# B&R Automation Studio project Stojan1
Automation Studio 4.2.9.65 SP

## Configuration Config1

CPU 5PPC2100.BY22-000, AutomationRuntime D4.26, Build 4.1.2, Vc V4.26.1

### Task classes (Cpu.sw)
```
Cyclic#1:
  ncsdcctrl <- ncsdcctrl.prg
  RdBlock_0 <- RdBlock_0.prg
Binaries: TCData, arconfig, asfw, ashwd, iomap, User, Role, sysconf
```

### IoMap.iom - 5PPC2100_BY22_000/IoMap.iom
```iecst
VAR_CONFIG
	::RdBlock_0:FltMtuRd[1] AT %IB."X20AP3131".RxByte1;
	::RdBlock_0:FltMtuRd[2] AT %IB."X20AP3131".RxByte2;
	::RdBlock_0:FltMtuRd[3] AT %IB."X20AP3131".RxByte3;
	::RdBlock_0:FltMtuRd[4] AT %IB."X20AP3131".RxByte4;
	::RdBlock_0:FltMtuRd[5] AT %IB."X20AP3131".RxByte5;
	::RdBlock_0:FltMtuRd[6] AT %IB."X20AP3131".RxByte6;
	::RdBlock_0:FltMtuRd[7] AT %IB."X20AP3131".RxByte7;
	::RdBlock_0:RBTrigDFT AT %IX."X20AP3131".RBTrigDFT;
	::RdBlock_0:TrigDFT AT %QX."X20AP3131".TrigDFT;
	::RdBlock_0:EnabEnergy AT %QX."X20AP3131".EnabEnergy;
	::RdBlock_0:FltMtuWr[0] AT %QB."X20AP3131".OutputSequence;
	RdBlock_0:FltMtuRd[0] AT %IB."X20AP3131".InputSequence;
END_VAR
```

## Configuration TestStand1

CPU , AutomationRuntime D3.10, Build 4.1.2

### Task classes (Cpu.sw)
```
Cyclic#1 (cycle 2000 us, tolerance 0 us):
  ncsdcctrl <- ncsdcctrl.prg
  RdBlock_0 <- RdBlock_0.prg
Cyclic#2 (cycle 20000 us, tolerance 20000 us):
  GearAxis01 <- Samples.GearAxis01.prg
  GearAxis02 <- Samples.GearAxis02.prg
DataObjects: Acp10sys
NcDataObjects: gAxis01a <- gAxis01obj.gAxis01a.dob, gAxis01i <- gAxis01obj.gAxis01i.dob, gAxis02a <- gAxis02obj.gAxis02a.dob, gAxis02i <- gAxis02obj.gAxis02i.dob, gAxis03a <- gAxis03obj.gAxis03a.dob, gAxis03i <- gAxis03obj.gAxis03i.dob, gAxis04a <- gAxis04obj.gAxis04a.dob, gAxis04i <- gAxis04obj.gAxis04i.dob
Binaries: ashwd, sysconf, asfw, arconfig, iomap, acp10map, acp10cfg
Libraries: Acp10_MC, brsystem, Acp10man, sys_lib, NcGlobal, Acp10par, Runtime, Acp10sdc, asstring, Acp10sim, astime, fileio, powerlnk, asieccon, asfltgen
```

### Hardware
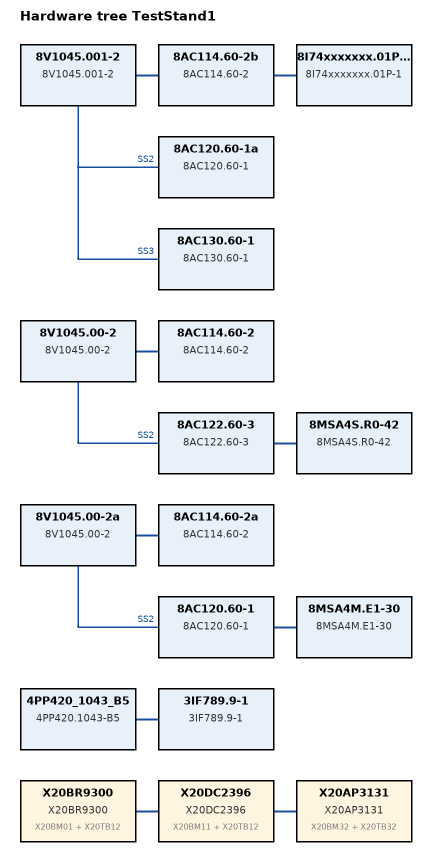
```
3IF789.9-1 : 3IF789.9-1 v1.1.3.1  [SS -> 4PP420_1043_B5.SS1]
  Connector IF2:
    EplEthInterfaceRedundant = 0
4PP420_1043_B5 : 4PP420.1043-B5 v1.0.0.0
  Connector IF5:
    ActivateDevice = 1
  TimerDeviceType = EPLX2X
  TimerDevice = 3IF789.9-1.IF2
  TaskClassIdleTime = 2000
  Cyclic1Duration = 2000
  Cyclic1Tolerance = 0
  Cyclic1Output = 1
  Cyclic2Duration = 20000
  Cyclic2Tolerance = 20000
  Cyclic3Duration = 50000
  Cyclic3Tolerance = 50000
  Cyclic4Duration = 100000
  Cyclic4Tolerance = 100000
  Cyclic5Duration = 200000
  Cyclic5Tolerance = 200000
  Cyclic6Duration = 500000
  Cyclic6Tolerance = 500000
  Cyclic7Duration = 1000000
  Cyclic7Tolerance = 1000000
  Cyclic8Duration = 10000
  Cyclic8Tolerance = 30000000
  EthernetHostName = stojan1
8AC114.60-2 : 8AC114.60-2 v1.0.0.8  [SS -> 8V1045.00-2.SS1; PLK1 -> 3IF789.9-1.IF2 (NodeNumber=1); PLK2 -> 8AC114.60-2a.PLK1 (NodeNumber=1)]
8AC114.60-2a : 8AC114.60-2 v1.0.0.8  [SS -> 8V1045.00-2a.SS1; PLK1 -> 8AC114.60-2.PLK2 (NodeNumber=2); PLK2 -> 8AC114.60-2b.PLK1 (NodeNumber=2)]
8AC114.60-2b : 8AC114.60-2 v1.0.0.8  [SS -> 8V1045.001-2.SS1; PLK1 -> 8AC114.60-2a.PLK2 (NodeNumber=3); PLK2 -> 8I74xxxxxxx.01P-1.PLK1 (NodeNumber=3)]
8AC120.60-1 : 8AC120.60-1 v1.0.0.2  [SS -> 8V1045.00-2a.SS2]
8AC120.60-1a : 8AC120.60-1 v1.0.0.2  [SS -> 8V1045.001-2.SS2]
8AC122.60-3 : 8AC122.60-3 v1.0.0.2  [SS -> 8V1045.00-2.SS2]
8AC130.60-1 : 8AC130.60-1 v1.0.0.3  [SS -> 8V1045.001-2.SS3]
8I74xxxxxxx.01P-1 : 8I74xxxxxxx.01P-1 v1.2.0.1  [PLK1 -> 8AC114.60-2b.PLK2 (NodeNumber=4)]
  Supervision = off
  CTT = 3
  AUT = 1
  NPR = 75
  COS = 80
  UNS = 400
  NCR = 19
  NSP = 1395
  RSA = 11302
  LFA = 4842
8MSA4M.E1-30 : 8MSA4M.E1-30 v1.0.0.0  [EC -> 8AC120.60-1.EC; MT -> 8V1045.00-2a.MT1]
8MSA4S.R0-42 : 8MSA4S.R0-42 v1.0.0.0  [EC -> 8AC122.60-3.EC; MT -> 8V1045.00-2.MT1]
8V1045.00-2 : 8V1045.00-2 v1.0.0.2
  BothEndSwitchesAreNormallyOpen_r1 = on
  QuickStopIsNormallyOpen_r1 = on
8V1045.00-2a : 8V1045.00-2 v1.0.0.2
  BothEndSwitchesAreNormallyOpen_r1 = on
  QuickStopIsNormallyOpen_r1 = on
8V1045.001-2 : 8V1045.001-2 v1.0.0.0
  BothEndSwitchesAreNormallyOpen_r1 = on
  QuickStopIsNormallyOpen_r1 = on
X20AP3131 : X20AP3131 v1.0.1.0  [SS1 -> X20TB32.SS; SL -> X20BM32.SL1]
  Supervision = off
  EnergyUnit = 1Ws
  VoltageLimit = off
  DisPFmeanT = off
  DisPmeanT = off
  DisQmeanT = off
  DisSmeanT = off
  DisAcEnT = off
  DisReacEnT = off
  DisAppEnT = off
  FlatStreamActivate = on
  InputMTU = 23byte
X20BM01 : X20BM01 v1.0.1.1
X20BM11 : X20BM11 v1.0.0.1  [X2X1 -> X20BM01.X2X2]
X20BM32 : X20BM32 v1.0.0.1  [X2X1 -> X20BM11.X2X2]
X20BR9300 : X20BR9300 v1.0.3.0  [SS1 -> X20TB12.SS; SL -> X20BM01.SL1; X2X1 -> 3IF789.9-1.IF1]
  Supervision = off
X20DC2396 : X20DC2396 v1.0.2.1  [SS1 -> X20TB12a.SS; SL -> X20BM11.SL1]
  Supervision = off
X20TB12 : X20TB12 v1.0.0.0
X20TB12a : X20TB12 v1.0.0.0
X20TB32 : X20TB32 v1.0.0.1
```

### IoMap.iom - 4PP420_1043_B5/IoMap.iom
```iecst
(********************************************************************
 * COPYRIGHT -- Bernecker + Rainer
 ********************************************************************
 * File: IoMap.iom
 * Author: necidj
 * Created: March 11, 2014
 ********************************************************************
 * IO mapping file
 ********************************************************************)
VAR_CONFIG
	Cyclic#1.gAxis04_DrvIf.iLifeCnt AT %IB."8I74xxxxxxx.01P-1".SDC_LifeCnt;
	Cyclic#1.gAxis04_DrvIf.iDrvOK AT %IX."8I74xxxxxxx.01P-1".ETAD_Input_Bool_02;
	Cyclic#1.gAxis04_DrvIf.oSetTime AT %QW."8I74xxxxxxx.01P-1".SDC_SetTime;
	Cyclic#1.gAxis04_DrvIf.oSetPos AT %QW."8I74xxxxxxx.01P-1".LFRD_Output;
	Cyclic#1.gAxis04_DiDoIf.iLifeCntDriveReady AT %IB."8I74xxxxxxx.01P-1".SDC_LifeCnt;
	Cyclic#1.gAxis04_DiDoIf.iLifeCntDriveEnable AT %IB."8I74xxxxxxx.01P-1".SDC_LifeCnt;
	Cyclic#1.gAxis04_DiDoIf.oDriveEnable AT %QX."8I74xxxxxxx.01P-1".CMDD_Output_Bool_00;
	Cyclic#1.gAxis04_ModuleOk AT %QX."8I74xxxxxxx.01P-1".CMDD_Output_Bool_01;
	Cyclic#1.gAxis04_ModuleOk AT %QX."8I74xxxxxxx.01P-1".CMDD_Output_Bool_02;
	Cyclic#1.gAxis04_ModuleOk AT %IX."8I74xxxxxxx.01P-1".ModuleOk;
	Cyclic#1.gAxis04_DiDoIf.oDriveEnable AT %QX."8I74xxxxxxx.01P-1".CMDD_Output_Bool_03;
	Cyclic#1.gAxis04_DiDoIf.iDriveReady AT %IX."8I74xxxxxxx.01P-1".ETAD_Input_Bool_02;
	gAxis04_DrvIf.oBrake AT %QX."8I74xxxxxxx.01P-1".OL1R_Output_Bool_02;
	gAxis04_EncIf.iActPos AT %IW."X20DC2396".Encoder01;
	gAxis04_EncIf.iEncOK AT %IX."X20DC2396".ModuleOk;
	::RdBlock_0:FltMtuRd[1] AT %IB."X20AP3131".RxByte1;
	::RdBlock_0:FltMtuRd[2] AT %IB."X20AP3131".RxByte2;
	::RdBlock_0:FltMtuRd[3] AT %IB."X20AP3131".RxByte3;
	::RdBlock_0:FltMtuRd[4] AT %IB."X20AP3131".RxByte4;
	::RdBlock_0:FltMtuRd[5] AT %IB."X20AP3131".RxByte5;
	::RdBlock_0:FltMtuRd[6] AT %IB."X20AP3131".RxByte6;
	::RdBlock_0:FltMtuRd[7] AT %IB."X20AP3131".RxByte7;
	::RdBlock_0:FltMtuRd[8] AT %IB."X20AP3131".RxByte8;
	::RdBlock_0:FltMtuRd[9] AT %IB."X20AP3131".RxByte9;
	::RdBlock_0:FltMtuRd[10] AT %IB."X20AP3131".RxByte10;
	::RdBlock_0:FltMtuRd[11] AT %IB."X20AP3131".RxByte11;
	::RdBlock_0:FltMtuRd[12] AT %IB."X20AP3131".RxByte12;
	::RdBlock_0:FltMtuRd[13] AT %IB."X20AP3131".RxByte13;
	::RdBlock_0:FltMtuRd[14] AT %IB."X20AP3131".RxByte14;
	::RdBlock_0:FltMtuRd[15] AT %IB."X20AP3131".RxByte15;
	::RdBlock_0:FltMtuRd[16] AT %IB."X20AP3131".RxByte16;
	::RdBlock_0:FltMtuRd[17] AT %IB."X20AP3131".RxByte17;
	::RdBlock_0:FltMtuRd[18] AT %IB."X20AP3131".RxByte18;
	::RdBlock_0:FltMtuRd[19] AT %IB."X20AP3131".RxByte19;
	::RdBlock_0:FltMtuRd[20] AT %IB."X20AP3131".RxByte20;
	::RdBlock_0:FltMtuRd[21] AT %IB."X20AP3131".RxByte21;
	::RdBlock_0:FltMtuRd[22] AT %IB."X20AP3131".RxByte22;
	::RdBlock_0:RBTrigDFT AT %IX."X20AP3131".RBTrigDFT;
	::RdBlock_0:TrigDFT AT %QX."X20AP3131".TrigDFT;
	::RdBlock_0:EnabEnergy AT %QX."X20AP3131".EnabEnergy;
	RdBlock_0:FltMtuRd[23]  AT %IB."X20AP3131".RxByte23;
	::RdBlock_0:FltMtuWr[0] AT %QB."X20AP3131".OutputSequence;
	RdBlock_0:FltMtuRd[0]  AT %IB."X20AP3131".InputSequence;
END_VAR
```

### Acp10cfg.ncc - 4PP420_1043_B5/Motion/Acp10cfg.ncc
```
NcConfiguration (Version=2.42.0, NcSwId=Acp10)
  ACP10CF1_typ:
    cnt_nettrc_rec_drive = 1500
    bufsize_trace_upload = 1200
    tc_nc_man_task = Cyclic #1
    glob_pv_as_ncobject = Yes
    ncsys_dl_broadcast = Yes
    ncsys_dl_acp_reset = Yes
    safemc_log_err_to_ax = Yes
    network_init:
      ncsw_init_execute = Yes
      automatic_execute = No
      node_nr_warning = Yes
      net_err_before_ncact = Yes
    nettrc:
      enter_parsecrec = Yes
      enter_ncaction = Yes
      save_ring_startidx = Yes
    cam_prof_download:
      cam_dat_dl_parallel = No
      tc_cam_dl_parallel = Task class for NC Manager task
    plk_if[0]:
      if_name = SL1.SS1.IF2
      tc_CycDat_PLCopen = Task class for NC Manager task
      mc_broadcast_extdat = No
    sdc_if[0]:
      if_name = SDC_IF1
      mc_broadcast_size = 800
      mc_broadcast_extdat = No
```

### Acp10map.ncm - 4PP420_1043_B5/Motion/Acp10map.ncm
```
NcMapping (NcSwId=Acp10)
  NcObject gAxis01 (ModuleId=8V1045.00-2, Type=ncAXIS, Channel=1, AcoposSimulation=Standard, InitParameter=gAxis01i, AcoposParameter=gAxis01a, Disabled=FALSE, ModuleDisabled=FALSE)
  NcObject 8V1045.00-2_ncV_AXIS1 (ModuleId=8V1045.00-2, Type=ncV_AXIS, Channel=1, Disabled=TRUE, ModuleDisabled=FALSE)
  NcObject gAxis02 (ModuleId=8V1045.00-2a, Type=ncAXIS, Channel=1, AcoposSimulation=Standard, InitParameter=gAxis02i, AcoposParameter=gAxis02a, Disabled=FALSE, ModuleDisabled=FALSE)
  NcObject 8V1045.00-2a_ncV_AXIS1 (ModuleId=8V1045.00-2a, Type=ncV_AXIS, Channel=1, Disabled=TRUE, ModuleDisabled=FALSE)
  NcObject gAxis03 (ModuleId=8V1045.001-2, Type=ncAXIS, Channel=1, AcoposSimulation=Off, InitParameter=gAxis03i, AcoposParameter=gAxis03a, Disabled=FALSE, ModuleDisabled=FALSE)
  NcObject 8V1045.001-2_ncV_AXIS1 (ModuleId=8V1045.001-2, Type=ncV_AXIS, Channel=1, Disabled=TRUE, ModuleDisabled=FALSE)
  NcObject gAxis04 (ModuleId=8I74xxxxxxx.01P-1, ModuleAddress=SDC_IF1.ST1, Type=ncAXIS, Channel=1, AcoposSimulation=Off, InitParameter=gAxis04i, AcoposParameter=gAxis04a, Disabled=FALSE, ModuleDisabled=FALSE)
```

## Logical view

Binary libraries used (declarations not repeated): operator, runtime, astime, AsIecCon, brsystem, sys_lib, asstring, Acp10man 2.43.1, Acp10par 2.43.1, NcGlobal 2.43.1, Acp10_MC 2.43.1, Acp10sdc 2.43.1, Acp10sim 2.43.1, AsFltGen

### Global.var - Global variables
```iecst
(********************************************************************
 * COPYRIGHT -- Bernecker + Rainer
 ********************************************************************
 * File: Global.var
 * Author: necidj
 * Created: March 11, 2014
 ********************************************************************
 * Global variables of project TestStandBasic
 ********************************************************************)
VAR
	gAxis01 : ACP10AXIS_typ;
	gAxis02 : ACP10AXIS_typ;
	gAxis03 : ACP10AXIS_typ;
	gAxis04 : ACP10AXIS_typ;
	gAxis04_HW : SdcHwCfg_typ := (0);
	gAxis04_EncIf : SdcEncIf16_typ := (0);
	gAxis04_DrvIf : SdcDrvIf16_typ := (0);
	gAxis04_DiDoIf : SdcDiDoIf_typ := (0);
	gAxis04_ModuleOk : BOOL := 0;
END_VAR
```


### Package Logical/gAxis01obj - gAxis01obj

- Data object Logical/gAxis01obj/gAxis01a (Apt) (no source held here)

### Data object Logical/gAxis01obj/gAxis01i (Ax)

#### gAxis01i.ax
```
InitParameter (Version=2.43.1, NcSwId=ACP10)
  ACP10AXIS_typ:
    dig_in:
      level:
        reference = ncACTIV_HI
        pos_hw_end = ncACTIV_HI
        neg_hw_end = ncACTIV_HI
        trigger1 = ncACTIV_HI
        trigger2 = ncACTIV_HI
    encoder_if:
      parameter:
        count_dir = ncSTANDARD
        scaling:
          load:
            units = 1000
            rev_motor = 1
    limit:
      parameter:
        v_pos = 10000.0
        v_neg = 10000.0
        a1_pos = 50000.0
        a2_pos = 50000.0
        a1_neg = 50000.0
        a2_neg = 50000.0
        t_jolt = 0.0
        t_in_pos = 0.0
        pos_sw_end = 8388607
        neg_sw_end = -8388608
        ds_warning = 500.0
        ds_stop = 1000.0
        a_stop = 1.0e+30
        dv_stop = 0.0
        dv_stop_mode = ncOFF
    controller:
      mode = ncPOSITION
      position:
        kv = 440.0
        tn = 0.0
        t_predict = 0.0004
        t_total = 0.0004
        p_max = 1.0e+30
        i_max = 0.0
      speed:
        kv = 3.5
        tn = 0.0
        t_filter = 0.0012
        isq_filter1:
          type = ncNOTCH
          a0 = 2485.32
          a1 = 400.0
          b0 = 0.0
          b1 = 0.0
          b2 = 0.0
          c0_par_id = 0
          c1_par_id = 0
        isq_filter2:
          type = ncOFF
          a0 = 0.0
          a1 = 0.0
          b0 = 0.0
          b1 = 0.0
          b2 = 0.0
          c0_par_id = 0
          c1_par_id = 0
        isq_filter3:
          type = ncOFF
          a0 = 0.0
          a1 = 0.0
          b0 = 0.0
          b1 = 0.0
          b2 = 0.0
          c0_par_id = 0
          c1_par_id = 0
      uf:
        type = ncLINEAR
        auto_config = ncMOTOR_PAR
        u0 = 0.0
        un = 0.0
        fn = 50.0
        k_f_slip = 0.0
      ff:
        torque_load = 0.0
        torque_pos = 0.0
        torque_neg = 0.0
        kv_torque = 0.0
        inertia = 0.0
        t_filter_a = 0.0
    move:
      stop:
        parameter[0]:
          decel_ramp = ncA_LIMIT
          controller = ncON
        parameter[1]:
          decel_ramp = ncA_LIMIT
          controller = ncON
        parameter[2]:
          decel_ramp = ncA_LIMIT
          controller = ncON
        parameter[3]:
          decel_ramp = ncA_LIMIT
          controller = ncON
        quickstop:
          decel_ramp = ncA_LIMIT
        drive_error:
          decel_ramp = ncA_LIMIT
      homing:
        parameter:
          s = 0
          v_switch = 5000.0
          v_trigger = 500.0
          a = 50000.0
          mode = ncDIRECT
          edge_sw = ncPOSITIVE
          start_dir = ncPOSITIVE
          trigg_dir = ncPOSITIVE
          ref_pulse = ncOFF
          fix_dir = ncOFF
          tr_s_block = 0.0
          torque_lim = 0.0
          ds_block = 0.0
          ds_stop = 0.0
      basis:
        parameter:
          v_pos = 5000.0
          v_neg = 5000.0
          a1_pos = 50000.0
          a2_pos = 50000.0
          a1_neg = 50000.0
          a2_neg = 50000.0
    message:
      text:
        parameter:
          format = ncBREAK
          columns = 80
          data_modul = acp10etxen
```

### Package Logical/gAxis02obj - gAxis02obj

### Data object Logical/gAxis02obj/gAxis02a (Apt)

#### gAxis02a.apt
```
AcoposParameterTable:
  Root Parameters
```

### Data object Logical/gAxis02obj/gAxis02i (Ax)

#### gAxis02i.ax
```
InitParameter (Version=2.43.1, NcSwId=ACP10)
  ACP10AXIS_typ:
    dig_in:
      level:
        reference = ncACTIV_HI
        pos_hw_end = ncACTIV_HI
        neg_hw_end = ncACTIV_HI
        trigger1 = ncACTIV_HI
        trigger2 = ncACTIV_HI
    encoder_if:
      parameter:
        count_dir = ncSTANDARD
        scaling:
          load:
            units = 1000
            rev_motor = 1
    limit:
      parameter:
        v_pos = 10000.0
        v_neg = 10000.0
        a1_pos = 50000.0
        a2_pos = 50000.0
        a1_neg = 50000.0
        a2_neg = 50000.0
        t_jolt = 0.0
        t_in_pos = 0.0
        pos_sw_end = 8388607
        neg_sw_end = -8388608
        ds_warning = 500.0
        ds_stop = 1000.0
        a_stop = 1.0e+30
        dv_stop = 0.0
        dv_stop_mode = ncOFF
    controller:
      mode = ncPOSITION
      position:
        kv = 40.0
        tn = 0.0
        t_predict = 0.0004
        t_total = 0.0004
        p_max = 1.0e+30
        i_max = 0.0
      speed:
        kv = 1.2
        tn = 0.0
        t_filter = 0.0004
        isq_filter1:
          type = ncNOTCH
          a0 = 1771.04
          a1 = 400.0
          b0 = 0.0
          b1 = 0.0
          b2 = 0.0
          c0_par_id = 0
          c1_par_id = 0
        isq_filter2:
          type = ncOFF
          a0 = 0.0
          a1 = 0.0
          b0 = 0.0
          b1 = 0.0
          b2 = 0.0
          c0_par_id = 0
          c1_par_id = 0
        isq_filter3:
          type = ncOFF
          a0 = 0.0
          a1 = 0.0
          b0 = 0.0
          b1 = 0.0
          b2 = 0.0
          c0_par_id = 0
          c1_par_id = 0
      uf:
        type = ncLINEAR
        auto_config = ncMOTOR_PAR
        u0 = 0.0
        un = 0.0
        fn = 50.0
        k_f_slip = 0.0
      ff:
        torque_load = 0.0
        torque_pos = 0.0
        torque_neg = 0.0
        kv_torque = 0.0
        inertia = 0.0
        t_filter_a = 0.0
    move:
      stop:
        parameter[0]:
          decel_ramp = ncA_LIMIT
          controller = ncON
        parameter[1]:
          decel_ramp = ncA_LIMIT
          controller = ncON
        parameter[2]:
          decel_ramp = ncA_LIMIT
          controller = ncON
        parameter[3]:
          decel_ramp = ncA_LIMIT
          controller = ncON
        quickstop:
          decel_ramp = ncA_LIMIT
        drive_error:
          decel_ramp = ncA_LIMIT
      homing:
        parameter:
          s = 0
          v_switch = 5000.0
          v_trigger = 500.0
          a = 50000.0
          mode = ncDIRECT
          edge_sw = ncPOSITIVE
          start_dir = ncPOSITIVE
          trigg_dir = ncPOSITIVE
          ref_pulse = ncOFF
          fix_dir = ncOFF
          tr_s_block = 0.0
          torque_lim = 0.0
          ds_block = 0.0
          ds_stop = 0.0
      basis:
        parameter:
          v_pos = 5000.0
          v_neg = 5000.0
          a1_pos = 50000.0
          a2_pos = 50000.0
          a1_neg = 50000.0
          a2_neg = 50000.0
    message:
      text:
        parameter:
          format = ncBREAK
          columns = 80
          data_modul = acp10etxen
```

### Package Logical/gAxis03obj - gAxis03obj

- Data object Logical/gAxis03obj/gAxis03a (Apt) (no source held here)

### Data object Logical/gAxis03obj/gAxis03i (Ax)

#### gAxis03i.ax
```
InitParameter (Version=2.42.1, NcSwId=ACP10)
  ACP10AXIS_typ:
    dig_in:
      level:
        reference = ncACTIV_HI
        pos_hw_end = ncACTIV_HI
        neg_hw_end = ncACTIV_HI
        trigger1 = ncACTIV_HI
        trigger2 = ncACTIV_HI
    encoder_if:
      parameter:
        count_dir = ncSTANDARD
        scaling:
          load:
            units = 1000
            rev_motor = 1
    limit:
      parameter:
        v_pos = 10000.0
        v_neg = 10000.0
        a1_pos = 50000.0
        a2_pos = 50000.0
        a1_neg = 50000.0
        a2_neg = 50000.0
        t_jolt = 0.0
        t_in_pos = 0.0
        pos_sw_end = 8388607
        neg_sw_end = -8388608
        ds_warning = 500.0
        ds_stop = 1000.0
        a_stop = 1.0e+30
        dv_stop = 0.0
        dv_stop_mode = ncOFF
    controller:
      mode = ncPOSITION + ncFF
      position:
        kv = 520.0
        tn = 0.0
        t_predict = 0.0004
        t_total = 0.0004
        p_max = 1.0e+30
        i_max = 0.0
      speed:
        kv = 0.2
        tn = 0.0
        t_filter = 0.0
        isq_filter1:
          type = ncOFF
          a0 = 0.0
          a1 = 0.0
          b0 = 0.0
          b1 = 0.0
          b2 = 0.0
          c0_par_id = 0
          c1_par_id = 0
        isq_filter2:
          type = ncOFF
          a0 = 0.0
          a1 = 0.0
          b0 = 0.0
          b1 = 0.0
          b2 = 0.0
          c0_par_id = 0
          c1_par_id = 0
        isq_filter3:
          type = ncOFF
          a0 = 0.0
          a1 = 0.0
          b0 = 0.0
          b1 = 0.0
          b2 = 0.0
          c0_par_id = 0
          c1_par_id = 0
      uf:
        type = ncLINEAR
        auto_config = ncMOTOR_PAR
        u0 = 0.0
        un = 0.0
        fn = 50.0
        k_f_slip = 0.0
      ff:
        torque_load = 0.0
        torque_pos = 0.0287764
        torque_neg = 0.0287767
        kv_torque = 0.00626887
        inertia = 0.00413145
        t_filter_a = 0.0
    move:
      stop:
        parameter[0]:
          decel_ramp = ncA_LIMIT
          controller = ncON
        parameter[1]:
          decel_ramp = ncA_LIMIT
          controller = ncON
        parameter[2]:
          decel_ramp = ncA_LIMIT
          controller = ncON
        parameter[3]:
          decel_ramp = ncA_LIMIT
          controller = ncON
        quickstop:
          decel_ramp = ncA_LIMIT
        drive_error:
          decel_ramp = ncA_LIMIT
      homing:
        parameter:
          s = 0
          v_switch = 5000.0
          v_trigger = 500.0
          a = 50000.0
          mode = ncDIRECT
          edge_sw = ncPOSITIVE
          start_dir = ncPOSITIVE
          trigg_dir = ncPOSITIVE
          ref_pulse = ncOFF
          fix_dir = ncOFF
          tr_s_block = 0.0
          torque_lim = 0.0
          ds_block = 0.0
          ds_stop = 0.0
      basis:
        parameter:
          v_pos = 5000.0
          v_neg = 5000.0
          a1_pos = 50000.0
          a2_pos = 50000.0
          a1_neg = 50000.0
          a2_neg = 50000.0
    message:
      text:
        parameter:
          format = ncBREAK
          columns = 80
          data_modul = acp10etxen
```

### Package Logical/gAxis04obj - gAxis04obj

### Data object Logical/gAxis04obj/gAxis04a (Apt)

#### gAxis04a.apt
```
AcoposParameterTable:
  Root Parameters:
    230 = PCTRL_S_SET (Name=PCTRL_S_ACT_PARID)
    64201 = 546116,666666667 (Name=SERVO_V_MAX_OUTPUT)
    90 = 77 (Name=BRAKE_MODE)  // Motor holding brake: Mode
```

### Data object Logical/gAxis04obj/gAxis04i (Ax)

#### gAxis04i.ax
```
InitParameter (Version=2.42.1, NcSwId=ACP10)
  ACP10AXIS_typ:
    dig_in:
      level:
        reference = ncACTIV_HI
        pos_hw_end = ncACTIV_HI
        neg_hw_end = ncACTIV_HI
        trigger1 = ncACTIV_HI
        trigger2 = ncACTIV_HI
    encoder_if:
      parameter:
        count_dir = ncSTANDARD
        scaling:
          load:
            units = 1000
            rev_motor = 1
    limit:
      parameter:
        v_pos = 10000.0
        v_neg = 10000.0
        a1_pos = 50000.0
        a2_pos = 50000.0
        a1_neg = 50000.0
        a2_neg = 50000.0
        t_jolt = 0.0
        t_in_pos = 0.0
        pos_sw_end = 8388607
        neg_sw_end = -8388608
        ds_warning = 500.0
        ds_stop = 1000.0
        a_stop = 1.0e+30
        dv_stop = 0.0
        dv_stop_mode = ncOFF
    controller:
      mode = ncPOSITION
      position:
        kv = 50.0
        tn = 0.0
        t_predict = 0.01
        t_total = 0.01
        p_max = 10000.0
        i_max = 0.0
      speed:
        kv = 2.0
        tn = 0.0
        t_filter = 0.0
        isq_filter1:
          type = ncOFF
          a0 = 0.0
          a1 = 0.0
          b0 = 0.0
          b1 = 0.0
          b2 = 0.0
          c0_par_id = 0
          c1_par_id = 0
        isq_filter2:
          type = ncOFF
          a0 = 0.0
          a1 = 0.0
          b0 = 0.0
          b1 = 0.0
          b2 = 0.0
          c0_par_id = 0
          c1_par_id = 0
        isq_filter3:
          type = ncOFF
          a0 = 0.0
          a1 = 0.0
          b0 = 0.0
          b1 = 0.0
          b2 = 0.0
          c0_par_id = 0
          c1_par_id = 0
      uf:
        type = ncLINEAR
        auto_config = ncMOTOR_PAR
        u0 = 0.0
        un = 0.0
        fn = 50.0
        k_f_slip = 0.0
      ff:
        torque_load = 0.0
        torque_pos = 0.0
        torque_neg = 0.0
        kv_torque = 0.0
        inertia = 0.0
        t_filter_a = 0.0
    move:
      stop:
        parameter[0]:
          decel_ramp = ncA_LIMIT
          controller = ncON
        parameter[1]:
          decel_ramp = ncA_LIMIT
          controller = ncON
        parameter[2]:
          decel_ramp = ncA_LIMIT
          controller = ncON
        parameter[3]:
          decel_ramp = ncA_LIMIT
          controller = ncON
        quickstop:
          decel_ramp = ncA_LIMIT
        drive_error:
          decel_ramp = ncA_LIMIT
      homing:
        parameter:
          s = 0
          v_switch = 5000.0
          v_trigger = 500.0
          a = 50000.0
          mode = ncDIRECT
          edge_sw = ncPOSITIVE
          start_dir = ncPOSITIVE
          trigg_dir = ncPOSITIVE
          ref_pulse = ncOFF
          fix_dir = ncOFF
          tr_s_block = 0.0
          torque_lim = 0.0
          ds_block = 0.0
          ds_stop = 0.0
      basis:
        parameter:
          v_pos = 5000.0
          v_neg = 5000.0
          a1_pos = 50000.0
          a2_pos = 50000.0
          a1_neg = 50000.0
          a2_neg = 50000.0
    message:
      text:
        parameter:
          format = ncBREAK
          columns = 80
          data_modul = acp10etxen
```

### Program Logical/ncsdcctrl (IEC)

#### ncsdcctrlCyclic.st
```iecst
(********************************************************************
 * COPYRIGHT -- Bernecker + Rainer
 ********************************************************************
 * Program: ncsdcctrl
 * File: ncsdcctrlCyclic.st
 * Author: necidj
 * Created: March 11, 2014
 ********************************************************************
 * Implementation of program ncsdcctrl
 ********************************************************************)

PROGRAM _CYCLIC

(* ### BEGIN gAxis04 ### *)

(* life counter emulation of digital inputs *)
 gAxis04_DiDoIf.iLifeCntReference := gAxis04_DiDoIf.iLifeCntReference + 1;
 gAxis04_DiDoIf.iLifeCntNegHwEnd  := gAxis04_DiDoIf.iLifeCntNegHwEnd  + 1;
 gAxis04_DiDoIf.iLifeCntPosHwEnd  := gAxis04_DiDoIf.iLifeCntPosHwEnd  + 1;

(* ### END gAxis04 ### *)

END_PROGRAM
```

#### ncsdcctrlInit.st
```iecst
(********************************************************************
 * COPYRIGHT -- Bernecker + Rainer
 ********************************************************************
 * Program: ncsdcctrl
 * File: ncsdcctrlInit.st
 * Author: necidj
 * Created: March 11, 2014
 ********************************************************************
 * Implementation of program ncsdcctrl
 ********************************************************************)

PROGRAM _INIT

(* ### BEGIN gAxis04 ### *)

(* initialize variables *)
 gAxis04_HW.DrvIf_Typ := ncSDC_DRVSERVO16;
 strcpy( ADR(gAxis04_HW.DrvIf_Name[0]), ADR('gAxis04_DrvIf') );
 gAxis04_HW.DiDoIf_Typ := ncSDC_DIDO;
 strcpy( ADR(gAxis04_HW.DiDoIf_Name[0]), ADR('gAxis04_DiDoIf') );

(* force variable offset generation *)
 gAxis04.size                      := gAxis04.size;
 gAxis04_DrvIf.iLifeCnt            := gAxis04_DrvIf.iLifeCnt;
 gAxis04_DiDoIf.iLifeCntDriveReady := gAxis04_DiDoIf.iLifeCntDriveReady;
 gAxis04_ModuleOk                  := gAxis04_ModuleOk;

(* assign your hardware inputs here*)

(* gAxis04_DiDoIf.iPosHwEnd  := gAxis04_DiDoIf.iPosHwEnd;
 gAxis04_DiDoIf.iNegHwEnd  := gAxis04_DiDoIf.iNegHwEnd;
 gAxis04_DiDoIf.iReference := gAxis04_DiDoIf.iReference;
 *)

(* ### END gAxis04 ### *)

END_PROGRAM
```

### Package Logical/Samples - Package

### Program Logical/Samples/GearAxis01 (IEC) - gear logical control

#### gearInit.st - init code
```iecst
PROGRAM _INIT

(* get axis object *)
Axis1Obj := ADR(gAxis01);  (*Master Axis*)
Axis2Obj := ADR(gAxis02);  (*Slave Axis*)

AxisStep := STATE_WAIT; (* start step *)

GearControl.Parameter.Velocity             := 1000; (*velocity for movement*)
GearControl.Parameter.Acceleration         := 5000; (*acceleration for movement*)
GearControl.Parameter.Deceleration         := 5000; (*deceleration for movement*)
GearControl.Parameter.JogVelocity          := 400;  (*velocity for jogging *)
GearControl.Parameter.RatioNumerator       := 1000; (*ratio numerator for coupling *)
GearControl.Parameter.RatioDenominator     := 1000; (*ratio denominator for coupling *)
END_PROGRAM
```

#### gear.var - Local variables
```iecst
VAR
	GearControl : gear_typ; (*control structure*)
	MC_GearIn_0 : MC_GearIn; (*Function Block*)
	MC_GearOut_0 : MC_GearOut; (*Function Block*)
	MC_Home_0 : MC_Home; (*Function Block*)
	MC_MoveAbsolute_0 : MC_MoveAbsolute; (*Function Block*)
	MC_MoveAdditive_0 : MC_MoveAdditive; (*Function Block*)
	MC_MoveVelocity_0 : MC_MoveVelocity; (*Function Block*)
	MC_Power_0 : MC_Power; (*Function Block*)
	MC_ReadActualPosition_0 : MC_ReadActualPosition; (*Function Block*)
	MC_ReadActualVelocity_0 : MC_ReadActualVelocity; (*Function Block*)
	MC_ReadAxisError_0 : MC_ReadAxisError; (*Function Block*)
	MC_ReadStatus_0 : MC_ReadStatus; (*Function Block*)
	MC_Reset_0 : MC_Reset; (*Function Block*)
	MC_Stop_0 : MC_Stop; (*Function Block*)
	MC_BR_ReadDriveStatus_0 : MC_BR_ReadDriveStatus; (*Function Block*)
	MC_Halt_0 : MC_Halt; (*Function Block*)
	Axis1Obj : UDINT; (*axis reference*)
	Axis2Obj : UDINT; (*axis reference*)
	AxisStep : UINT; (*current step in the step sequence*)
END_VAR
VAR CONSTANT
	STATE_POWER_ON : USINT := 1; (*constant for the step in which the controller is switched on*)
	STATE_MOVE_VELOCITY : USINT := 16; (*constant for the step in which a movement with defiened velocity is started*)
	STATE_MOVE_ADDITIVE : USINT := 15; (*constant for the step in which a movement with defiened distance is started*)
	STATE_READY : USINT := 10; (*constant for a waiting step*)
	STATE_JOG_NEGATIVE : USINT := 13; (*constant for the step in which a negative jogging movement is executed*)
	STATE_WAIT : USINT := 0; (* constant for a waiting step*)
	STATE_STOP : USINT := 11; (*constant for the step in which movements are stopped*)
	STATE_MOVE_ABSOLUTE : USINT := 14; (*constant for the step in which a movement to defiened position is started*)
	STATE_GEAR_START : USINT := 20; (*constant for the step in which the coupling is startet*)
	STATE_ERROR_RESET : USINT := 102; (*constant for the step in which the errors are reset*)
	STATE_ERROR_AXIS : USINT := 100; (*constant for the axis error step*)
	STATE_GEAR_STOP : USINT := 21; (*constant for the step in which the coupling is stopped*)
	STATE_JOG_POSITIVE : USINT := 12; (*constant for the step in which a positive jogging movement is executed*)
	STATE_ERROR : USINT := 101; (*constant for the error step*)
	STATE_HOME : USINT := 2; (*constant for the step in which the axis is homed*)
	STATE_HALT : USINT := 17; (*constant for the step in which movements are stopped*)
END_VAR
```

### Program Logical/Samples/GearAxis02 (IEC) - gear logical control

#### gear.typ
```iecst
TYPE
	gear_command_typ : 	STRUCT  (*command structure*)
		Power : BOOL; (*switch on the controller*)
		Home : BOOL; (*reference the axis*)
		MoveAbsolute : BOOL; (*move to an defined position*)
		MoveAdditive : BOOL; (*move a defiened distance*)
		MoveVelocity : BOOL; (*start a movement with a defiened velocity*)
		Halt : BOOL; (*stop every active movement*)
		Stop : BOOL; (*stop every active movement as long as is set*)
		MoveJogPos : BOOL; (*move in positive direction as long as is set*)
		MoveJogNeg : BOOL; (*move in negative direction as long as is set*)
		StartSlave : BOOL; (*start coupling beetween master and slave*)
		DisengageSlave : BOOL; (*stop coupling between master and slave*)
		ErrorAcknowledge : BOOL; (*reset active errors*)
	END_STRUCT;
	gear_parameter_typ : 	STRUCT  (*parameter structure*)
		Position : REAL; (*target-position for MoveAbsolute-Command*)
		Distance : REAL; (*distance for MoveAdditive-Command*)
		Velocity : REAL; (*velocity for MoveVelocity-Command*)
		Direction : USINT; (*direction for commanded movements*)
		Acceleration : REAL; (*acceleration for commanded movements*)
		Deceleration : REAL; (*deceleration for commanded movements*)
		HomePosition : REAL; (*target-position for referencing the axis*)
		HomeMode : USINT; (*homing mode*)
		JogVelocity : REAL; (*velocity for jogging movement*)
		RatioNumerator : INT; (*ratio numerator for coupling*)
		RatioDenominator : UINT; (*ratio denominator for coupling*)
	END_STRUCT;
	gear_status_typ : 	STRUCT  (*status structure*)
		ErrorID : UINT; (*ErrorID of any occured error*)
		ErrorText : ARRAY[0..3] OF STRING[79]; (*Error Text*)
		ActPosition : REAL; (*actual position of the axis*)
		ActVelocity : REAL; (*actual velocity of the axis*)
		DriveStatus : MC_DRIVESTATUS_TYP; (*actual status of the axis*)
	END_STRUCT;
	gear_axisState_typ : 	STRUCT  (*axis state structure*)
		Disabled : BOOL; (*if set, axis is in state Disabled*)
		StandStill : BOOL; (*if set, axis is in state StandsStill*)
		Homing : BOOL; (*if set, axis is in state Homing*)
		Stopping : BOOL; (*if set, axis is in state Stopping*)
		DiscreteMotion : BOOL; (*if set, axis is in state DiscreteMotion*)
		ContinuousMotion : BOOL; (*if set, axis is in state ContinuousMotion*)
		SynchronizedMotion : BOOL; (*if set, axis is in state SynchronizedMotion*)
		ErrorStop : BOOL; (*if set, axis is in state ErrorStop*)
	END_STRUCT;
	gear_typ : 	STRUCT  (*control structure*)
		Command : gear_command_typ; (*command structure*)
		Parameter : gear_parameter_typ; (*parameter structure*)
		Status : gear_status_typ; (*status structure*)
		AxisState : gear_axisState_typ; (*axis state structure*)
	END_STRUCT;
END_TYPE
```

#### gearCyclic.st
```iecst
(********************************************************************
 * COPYRIGHT -- Bernecker + Rainer
 ********************************************************************
 * PROGRAM: Gear
 * File: gearCyclic.st
 * Author: Bernecker + Rainer
 * Created: December 01, 2009
 ********************************************************************
 * Implementation of Program Gear
 ********************************************************************)
PROGRAM _CYCLIC

(***************************************************************
        Control Sequence
***************************************************************)

(* status information is read before the step sequencer to attain a shorter reaction time *)
(************************ MC_READSTATUS *************************)
MC_ReadStatus_0.Enable := NOT(MC_ReadStatus_0.Error);
MC_ReadStatus_0.Axis := Axis2Obj;
MC_ReadStatus_0();
GearControl.AxisState.Disabled             := MC_ReadStatus_0.Disabled;
GearControl.AxisState.StandStill           := MC_ReadStatus_0.StandStill;
GearControl.AxisState.Stopping             := MC_ReadStatus_0.Stopping;
GearControl.AxisState.Homing               := MC_ReadStatus_0.Homing;
GearControl.AxisState.DiscreteMotion       := MC_ReadStatus_0.DiscreteMotion;
GearControl.AxisState.ContinuousMotion     := MC_ReadStatus_0.ContinuousMotion;
GearControl.AxisState.SynchronizedMotion   := MC_ReadStatus_0.SynchronizedMotion;
GearControl.AxisState.ErrorStop            := MC_ReadStatus_0.Errorstop;

(********************MC_BR_READDRIVESTATUS***********************)
MC_BR_ReadDriveStatus_0.Enable := NOT(MC_BR_ReadDriveStatus_0.Error);
MC_BR_ReadDriveStatus_0.Axis := Axis2Obj;
MC_BR_ReadDriveStatus_0.AdrDriveStatus := ADR(GearControl.Status.DriveStatus);
MC_BR_ReadDriveStatus_0();

(******************** MC_READACTUALPOSITION *********************)
MC_ReadActualPosition_0.Enable := (NOT(MC_ReadActualPosition_0.Error));
MC_ReadActualPosition_0.Axis := Axis2Obj;
MC_ReadActualPosition_0();
IF(MC_ReadActualPosition_0.Valid = TRUE)THEN
    GearControl.Status.ActPosition := MC_ReadActualPosition_0.Position;
END_IF

(******************** MC_READACTUALVELOCITY *********************)
MC_ReadActualVelocity_0.Enable := (NOT(MC_ReadActualVelocity_0.Error));
MC_ReadActualVelocity_0.Axis := Axis2Obj;
MC_ReadActualVelocity_0();
IF(MC_ReadActualVelocity_0.Valid = TRUE)THEN
    GearControl.Status.ActVelocity := MC_ReadActualVelocity_0.Velocity;
END_IF

(************************ MC_READAXISERROR **********************)
MC_ReadAxisError_0.Enable := NOT(MC_ReadAxisError_0.Error);
MC_ReadAxisError_0.Axis := Axis2Obj;
MC_ReadAxisError_0.DataAddress := ADR(GearControl.Status.ErrorText);
MC_ReadAxisError_0.DataLength := SIZEOF(GearControl.Status.ErrorText);
MC_ReadAxisError_0.DataObjectName := 'acp10etxen';
MC_ReadAxisError_0();

(**************** CHECK FOR GENERAL AXIS ERROR ******************)
    IF ((MC_ReadAxisError_0.AxisErrorID <> 0) AND (MC_ReadAxisError_0.Valid = TRUE)) THEN
        AxisStep := STATE_ERROR_AXIS;
(***************** CHECK IF POWER SHOULD BE OFF *******************)
    ELSIF ((GearControl.Command.Power = FALSE) AND (MC_ReadAxisError_0.Valid = TRUE)) THEN
        IF ((MC_ReadStatus_0.Errorstop = TRUE) AND (MC_ReadStatus_0.Valid = TRUE)) THEN
            AxisStep := STATE_ERROR_RESET;
        ELSE
            AxisStep := STATE_WAIT;
        END_IF
    END_IF

(* central monitoring OF stop command attains a shorter reaction TIME in CASE OF emergency stop *)
(******************CHECK FOR STOP COMMAND************************)
    IF (GearControl.Command.Stop = TRUE) THEN
        IF ((AxisStep >= STATE_READY) AND (AxisStep <= STATE_ERROR)) THEN
            (* reset all fb execute inputs we use *)
            MC_Home_0.Execute := FALSE;
            MC_Stop_0.Execute := FALSE;
            MC_MoveAbsolute_0.Execute := FALSE;
            MC_MoveAdditive_0.Execute := FALSE;
            MC_MoveVelocity_0.Execute := FALSE;
            MC_GearIn_0.Execute := FALSE;
            MC_GearOut_0.Execute := FALSE;
            MC_Halt_0.Execute := FALSE;
            MC_ReadAxisError_0.Acknowledge := FALSE;
            MC_Reset_0.Execute := FALSE;

            (* reset user commands *)
            GearControl.Command.Halt := FALSE;
            GearControl.Command.Home := FALSE;
            GearControl.Command.MoveJogPos := FALSE;
            GearControl.Command.MoveJogNeg := FALSE;
            GearControl.Command.MoveVelocity := FALSE;
            GearControl.Command.MoveAbsolute := FALSE;
            GearControl.Command.MoveAdditive := FALSE;
            GearControl.Command.DisengageSlave := FALSE;
            GearControl.Command.StartSlave := FALSE;

            AxisStep := STATE_STOP;
        END_IF
    END_IF

CASE AxisStep OF

(******************** WAIT *************************)
    STATE_WAIT:  (* STATE: Wait *)
        IF (GearControl.Command.Power = TRUE) THEN
            AxisStep := STATE_POWER_ON;
        ELSE
            MC_Power_0.Enable := FALSE;
        END_IF

        (* reset all fb execute inputs we use *)
        MC_Home_0.Execute := FALSE;
        MC_Stop_0.Execute := FALSE;
        MC_MoveAbsolute_0.Execute := FALSE;
        MC_MoveAdditive_0.Execute := FALSE;
        MC_MoveVelocity_0.Execute := FALSE;
        MC_GearIn_0.Execute := FALSE;
        MC_GearOut_0.Execute := FALSE;
        MC_ReadAxisError_0.Acknowledge := FALSE;
        MC_Reset_0.Execute := FALSE;

        (* reset user commands *)
        GearControl.Command.Stop := FALSE;
        GearControl.Command.Home := FALSE;
        GearControl.Command.MoveJogPos := FALSE;
        GearControl.Command.MoveJogNeg := FALSE;
        GearControl.Command.MoveVelocity := FALSE;
        GearControl.Command.MoveAbsolute := FALSE;
        GearControl.Command.MoveAdditive := FALSE;
        GearControl.Command.DisengageSlave := FALSE;
        GearControl.Command.StartSlave := FALSE;

        GearControl.Status.ErrorID := 0;

(******************** POWER ON **********************)
    STATE_POWER_ON:  (* STATE: Power on *)
        MC_Power_0.Enable := TRUE;
        IF (MC_Power_0.Status = TRUE) THEN
            AxisStep := STATE_READY;
        END_IF
        (* if a power error occured go to error state *)
        IF (MC_Power_0.Error = TRUE) THEN
            GearControl.Status.ErrorID := MC_Power_0.ErrorID;
            AxisStep := STATE_ERROR;
        END_IF

(******************** READY **********************)
    STATE_READY:  (* STATE: Waiting for commands *)
        IF (GearControl.Command.Home = TRUE)THEN
            GearControl.Command.Home := FALSE;
            AxisStep := STATE_HOME;

        ELSIF (GearControl.Command.Stop = TRUE) THEN
            AxisStep := STATE_STOP;

        ELSIF (GearControl.Command.MoveJogPos = TRUE) THEN
            AxisStep := STATE_JOG_POSITIVE;

        ELSIF (GearControl.Command.MoveJogNeg = TRUE) THEN
            AxisStep := STATE_JOG_NEGATIVE;

        ELSIF (GearControl.Command.MoveAbsolute = TRUE) THEN
            GearControl.Command.MoveAbsolute := FALSE;
            AxisStep := STATE_MOVE_ABSOLUTE;

        ELSIF (GearControl.Command.MoveAdditive = TRUE) THEN
            GearControl.Command.MoveAdditive := FALSE;
            AxisStep := STATE_MOVE_ADDITIVE;

        ELSIF (GearControl.Command.MoveVelocity = TRUE) THEN
            GearControl.Command.MoveVelocity := FALSE;
            AxisStep := STATE_MOVE_VELOCITY;

        ELSIF (GearControl.Command.StartSlave = TRUE) THEN
            GearControl.Command.StartSlave := FALSE;
            AxisStep := STATE_GEAR_START;

        ELSIF (GearControl.Command.Halt = TRUE) THEN
            GearControl.Command.Halt := FALSE;
            AxisStep := STATE_HALT;
        END_IF

(******************** HOME **********************)
    STATE_HOME: (* STATE: start homing process *)
        MC_Home_0.Position := GearControl.Parameter.HomePosition;
        MC_Home_0.HomingMode := GearControl.Parameter.HomeMode;
        MC_Home_0.Execute := TRUE;
        IF (MC_Home_0.Done = TRUE) THEN
            MC_Home_0.Execute := FALSE;
            AxisStep := STATE_READY;
        END_IF
        (* if a homing error occured go to error state *)
        IF (MC_Home_0.Error = TRUE) THEN
            MC_Home_0.Execute := FALSE;
            GearControl.Status.ErrorID := MC_Home_0.ErrorID;
            AxisStep := STATE_ERROR;
        END_IF

(***********************HALT_MOVEMENT***************************)
    STATE_HALT:   (* STATE: Halt movement *)
        MC_Halt_0.Deceleration := GearControl.Parameter.Deceleration;
        MC_Halt_0.Execute := TRUE;
        IF (MC_Halt_0.Done = TRUE) THEN
            MC_Halt_0.Execute := FALSE;
            AxisStep := STATE_READY;
        END_IF
        (* check if error occured *)
        IF (MC_Halt_0.Error = TRUE) THEN
            GearControl.Status.ErrorID := MC_Halt_0.ErrorID;
            MC_Halt_0.Execute := FALSE;
            AxisStep := STATE_ERROR;
        END_IF

(*********************** STOP MOVEMENT *************************)
    STATE_STOP: (* STATE: Stop movement *)
        MC_Stop_0.Deceleration := GearControl.Parameter.Deceleration;
        MC_Stop_0.Execute := TRUE;
        (* if axis is stopped go to ready state *)
        IF ((MC_Stop_0.Done = TRUE) AND (GearControl.Command.Stop = FALSE)) THEN
             MC_Stop_0.Execute := FALSE;
             AxisStep := STATE_READY;
        END_IF
        (* check if error occured *)
        IF (MC_Stop_0.Error = TRUE) THEN
            GearControl.Status.ErrorID := MC_Stop_0.ErrorID;
            MC_Stop_0.Execute := FALSE;
            AxisStep := STATE_ERROR;
        END_IF

(******************** START JOG MOVEMENT POSITVE **********************)
    STATE_JOG_POSITIVE: (* STATE: Start jog movement in positive direction *)
        MC_MoveVelocity_0.Velocity      := GearControl.Parameter.JogVelocity;
        MC_MoveVelocity_0.Acceleration  := GearControl.Parameter.Acceleration;
        MC_MoveVelocity_0.Deceleration  := GearControl.Parameter.Deceleration;
        MC_MoveVelocity_0.Direction     := mcPOSITIVE_DIR;
        MC_MoveVelocity_0.Execute := TRUE;
        IF (GearControl.Command.MoveJogPos = FALSE) THEN
            MC_MoveVelocity_0.Execute := FALSE;
            AxisStep := STATE_HALT;
        END_IF
        (* check if error occured *)
        IF (MC_MoveVelocity_0.Error = TRUE) THEN
            GearControl.Status.ErrorID := MC_MoveVelocity_0.ErrorID;
            MC_MoveVelocity_0.Execute := FALSE;
            AxisStep := STATE_ERROR;
        END_IF

(******************** START JOG MOVEMENT NEGATIVE **********************)
    STATE_JOG_NEGATIVE: (* STATE: Start jog movement in negative direction *)
        MC_MoveVelocity_0.Velocity      := GearControl.Parameter.JogVelocity;
        MC_MoveVelocity_0.Acceleration  := GearControl.Parameter.Acceleration;
        MC_MoveVelocity_0.Deceleration  := GearControl.Parameter.Deceleration;
        MC_MoveVelocity_0.Direction     := mcNEGATIVE_DIR;
        MC_MoveVelocity_0.Execute := TRUE;
        IF (GearControl.Command.MoveJogNeg = FALSE) THEN
            MC_MoveVelocity_0.Execute := FALSE;
            AxisStep := STATE_HALT;
        END_IF
        (* check if error occured *)
        IF (MC_MoveVelocity_0.Error = TRUE) THEN
            GearControl.Status.ErrorID := MC_MoveVelocity_0.ErrorID;
            MC_MoveVelocity_0.Execute := FALSE;
            AxisStep := STATE_ERROR;
        END_IF

(******************** START ABSOLUTE MOVEMENT **********************)
    STATE_MOVE_ABSOLUTE: (* STATE: Start absolute movement *)
        MC_MoveAbsolute_0.Position      := GearControl.Parameter.Position;
        MC_MoveAbsolute_0.Velocity      := GearControl.Parameter.Velocity;
        MC_MoveAbsolute_0.Acceleration  := GearControl.Parameter.Acceleration;
        MC_MoveAbsolute_0.Deceleration  := GearControl.Parameter.Deceleration;
        MC_MoveAbsolute_0.Direction     := GearControl.Parameter.Direction;
        MC_MoveAbsolute_0.Execute := TRUE;
        (* check if commanded position is reached *)
        IF (GearControl.Command.Halt) THEN
            GearControl.Command.Halt := FALSE;
            MC_MoveAbsolute_0.Execute := FALSE;
            AxisStep := STATE_HALT;
        ELSIF (MC_MoveAbsolute_0.Done = TRUE) THEN
            MC_MoveAbsolute_0.Execute := FALSE;
            AxisStep := STATE_READY;
        END_IF
        (* check if error occured *)
        IF (MC_MoveAbsolute_0.Error = TRUE) THEN
            GearControl.Status.ErrorID := MC_MoveAbsolute_0.ErrorID;
            MC_MoveAbsolute_0.Execute := FALSE;
            AxisStep := STATE_ERROR;
        END_IF

(******************** START ADDITIVE MOVEMENT **********************)
    STATE_MOVE_ADDITIVE: (* STATE: Start additive movement *)
        MC_MoveAdditive_0.Distance      := GearControl.Parameter.Distance;
        MC_MoveAdditive_0.Velocity      := GearControl.Parameter.Velocity;
        MC_MoveAdditive_0.Acceleration  := GearControl.Parameter.Acceleration;
        MC_MoveAdditive_0.Deceleration  := GearControl.Parameter.Deceleration;
        MC_MoveAdditive_0.Execute := TRUE;
        (* check if commanded distance is reached *)
        IF (GearControl.Command.Halt) THEN
            GearControl.Command.Halt := FALSE;
            MC_MoveAdditive_0.Execute := FALSE;
            AxisStep := STATE_HALT;
        ELSIF (MC_MoveAdditive_0.Done = TRUE) THEN
            MC_MoveAdditive_0.Execute := FALSE;
            AxisStep := STATE_READY;
        END_IF
        (* check if error occured *)
        IF (MC_MoveAdditive_0.Error = TRUE) THEN
            GearControl.Status.ErrorID := MC_MoveAdditive_0.ErrorID;
            MC_MoveAdditive_0.Execute := FALSE;
            AxisStep := STATE_ERROR;
        END_IF

(******************** START VELOCITY MOVEMENT **********************)
    STATE_MOVE_VELOCITY: (* STATE: Start velocity movement *)
        MC_MoveVelocity_0.Velocity      := GearControl.Parameter.Velocity;
        MC_MoveVelocity_0.Acceleration  := GearControl.Parameter.Acceleration;
        MC_MoveVelocity_0.Deceleration  := GearControl.Parameter.Deceleration;
        MC_MoveVelocity_0.Direction	    := GearControl.Parameter.Direction;
        MC_MoveVelocity_0.Execute := TRUE;
        (* check if commanded velocity is reached *)
        IF (GearControl.Command.Halt) THEN
            GearControl.Command.Halt := FALSE;
            MC_MoveVelocity_0.Execute := FALSE;
            AxisStep := STATE_HALT;
        ELSIF (MC_MoveVelocity_0.InVelocity = TRUE) THEN
            MC_MoveVelocity_0.Execute := FALSE;
            AxisStep := STATE_READY;
        END_IF
        (* check if error occured *)
        IF (MC_MoveVelocity_0.Error = TRUE) THEN
            GearControl.Status.ErrorID := MC_MoveVelocity_0.ErrorID;
            MC_MoveVelocity_0.Execute := FALSE;
            AxisStep := STATE_ERROR;
        END_IF

(******************** START GEAR MOVEMENT **********************)
    STATE_GEAR_START: (* STATE: Start electronic gear coupling *)
        MC_GearIn_0.RatioNumerator  := GearControl.Parameter.RatioNumerator;
        MC_GearIn_0.RatioDenominator:= GearControl.Parameter.RatioDenominator;
        MC_GearIn_0.Acceleration    := GearControl.Parameter.Acceleration;
        MC_GearIn_0.Deceleration    := GearControl.Parameter.Deceleration;
        MC_GearIn_0.Execute := TRUE;
        (* wait for gear stop *)
        IF (GearControl.Command.Halt) THEN
            GearControl.Command.Halt := FALSE;
            MC_GearIn_0.Execute := FALSE;
            AxisStep := STATE_HALT;
        ELSIF (GearControl.Command.DisengageSlave = TRUE) THEN
            GearControl.Command.DisengageSlave := FALSE;
            MC_GearIn_0.Execute := FALSE;
            AxisStep := STATE_GEAR_STOP;
        END_IF
        (* check if error occured *)
        IF (MC_GearIn_0.Error = TRUE) THEN
            GearControl.Status.ErrorID := MC_GearIn_0.ErrorID;
            MC_GearIn_0.Execute := FALSE;
            AxisStep := STATE_ERROR;
        END_IF

(******************** STOP GEAR MOVEMENT **********************)
    STATE_GEAR_STOP: (* STATE: Stop electronic gear coupling *)
        MC_GearOut_0.Execute := TRUE;
        (* check if coupling is stopped *)
        IF (MC_GearOut_0.Done = TRUE) THEN
            MC_GearOut_0.Execute := FALSE;
            AxisStep := STATE_READY;
        END_IF
        (* check if error occured *)
        IF (MC_GearOut_0.Error = TRUE) THEN
            GearControl.Status.ErrorID := MC_GearOut_0.ErrorID;
            MC_GearOut_0.Execute := FALSE;
            AxisStep := STATE_ERROR;
        END_IF

(******************** FB-ERROR OCCURED *************************)
    STATE_ERROR: (* STATE: Error *)
        (* check if FB indicates an axis error *)
        IF (MC_ReadAxisError_0.AxisErrorCount<>0) THEN
            AxisStep := STATE_ERROR_AXIS;
        ELSE
            IF (GearControl.Command.ErrorAcknowledge = TRUE) THEN
                GearControl.Command.ErrorAcknowledge := FALSE;
                GearControl.Status.ErrorID := 0;
                (* reset axis if it is in axis state ErrorStop *)
                IF ((MC_ReadStatus_0.Errorstop = TRUE) AND (MC_ReadStatus_0.Valid = TRUE)) THEN
                    AxisStep := STATE_ERROR_RESET;
                ELSE
                    AxisStep := STATE_WAIT;
                END_IF
            END_IF
        END_IF

(******************** AXIS-ERROR OCCURED *************************)
    STATE_ERROR_AXIS: (* STATE: Axis Error *)
        IF (MC_ReadAxisError_0.Valid = TRUE) THEN
            IF (MC_ReadAxisError_0.AxisErrorID <> 0) THEN
                GearControl.Status.ErrorID := MC_ReadAxisError_0.AxisErrorID;
            END_IF
            MC_ReadAxisError_0.Acknowledge := FALSE;
            IF (GearControl.Command.ErrorAcknowledge = TRUE) THEN
                GearControl.Command.ErrorAcknowledge := FALSE;
                (* acknowledge axis error *)
                IF (MC_ReadAxisError_0.AxisErrorID <> 0) THEN
                    MC_ReadAxisError_0.Acknowledge := TRUE;
                END_IF
            END_IF
            IF (MC_ReadAxisError_0.AxisErrorCount = 0) THEN
                (* reset axis if it is in axis state ErrorStop *)
                GearControl.Status.ErrorID := 0;
                IF ((MC_ReadStatus_0.Errorstop = TRUE) AND (MC_ReadStatus_0.Valid = TRUE)) THEN
                    AxisStep := STATE_ERROR_RESET;
                ELSE
                    AxisStep := STATE_WAIT;
                END_IF
            END_IF
        END_IF

(******************** RESET DONE *************************)
    STATE_ERROR_RESET: (* STATE: Wait for reset done *)
        MC_Reset_0.Execute := TRUE;
        (* reset MC_Power.Enable if this FB is in Error*)
        IF (MC_Power_0.Error = TRUE) THEN
            MC_Power_0.Enable := FALSE;
        END_IF
        IF(MC_Reset_0.Done = TRUE)THEN
            MC_Reset_0.Execute := FALSE;
            AxisStep := STATE_WAIT;
        ELSIF(MC_Reset_0.Error = TRUE) THEN
            MC_Reset_0.Execute := FALSE;
            AxisStep := STATE_ERROR;
        END_IF
(******************** SEQUENCE END *************************)
END_CASE

(***************************************************************
        Function Block Calls
***************************************************************)

(************************** MC_POWER ****************************)
MC_Power_0.Axis := Axis2Obj; (* pointer to axis *)
MC_Power_0();

(************************** MC_HOME *****************************)
MC_Home_0.Axis := Axis2Obj;
MC_Home_0();

(********************** MC_MOVEABSOLUTE *************************)
MC_MoveAbsolute_0.Axis := Axis2Obj;
MC_MoveAbsolute_0();

(********************** MC_MOVEADDITIVE *************************)
MC_MoveAdditive_0.Axis := Axis2Obj;
MC_MoveAdditive_0();

(********************** MC_MOVEVELOCITY *************************)
MC_MoveVelocity_0.Axis := Axis2Obj;
MC_MoveVelocity_0();

(********************** MC_GEARIN *************************)
MC_GearIn_0.Master := Axis1Obj;
MC_GearIn_0.Slave := Axis2Obj;
MC_GearIn_0();

(********************** MC_GEAROUT *************************)
MC_GearOut_0.Slave := Axis2Obj;
MC_GearOut_0();

(************************** MC_STOP *****************************)
MC_Stop_0.Axis := Axis2Obj;
MC_Stop_0();

(**************************MC_HALT*******************************)
MC_Halt_0.Axis := Axis2Obj;
MC_Halt_0();

(************************** MC_RESET ****************************)
MC_Reset_0.Axis := Axis2Obj;
MC_Reset_0();

END_PROGRAM
```

#### gearInit.st
```iecst
PROGRAM _INIT

(* get axis object *)
Axis1Obj := ADR(gAxis02);  (*Master Axis*)
Axis2Obj := ADR(gAxis01);  (*Slave Axis*)

AxisStep := STATE_WAIT; (* start step *)

GearControl.Parameter.Velocity             := 1000; (*velocity for movement*)
GearControl.Parameter.Acceleration         := 5000; (*acceleration for movement*)
GearControl.Parameter.Deceleration         := 5000; (*deceleration for movement*)
GearControl.Parameter.JogVelocity          := 400;  (*velocity for jogging *)
GearControl.Parameter.RatioNumerator       := 1000; (*ratio numerator for coupling *)
GearControl.Parameter.RatioDenominator     := 1000; (*ratio denominator for coupling *)
END_PROGRAM
```

### Program Logical/RdBlock_0 (ANSIC) - cteni dat z X20AP karty

#### RdBlock_0.c - Implementation code
```c
/********************************************************************
 * COPYRIGHT -- Bernecker + Rainer
 ********************************************************************/

#include <bur/plctypes.h>
#include <AsDefault.h>
#include "AsFltGen.h"

#include "APMap.h"

// Variables for Flat Stream Interface to get whole X20AP31x1 Map

_LOCAL	 BOOL	 	Flt_Enable;
_LOCAL	 struct		fltRead	sFltRead;
_LOCAL	 struct		fltWrite sFltWrite;
_LOCAL	 X20AP31x1 	ApData;
_LOCAL	 SINT		TmpBuf[sizeof(X20AP31x1) + 16];
_LOCAL 	 USINT		BlockNum;
_LOCAL   UINT		BlockAct;
_LOCAL	DINT	ActiveEnergy;

void _INIT TestINIT( void )
{
	BlockNum = BlockAct = 0;
	Flt_Enable =  EnabEnergy = 1;

}

void _CYCLIC TestCYCLIC( void )
{
	ActiveEnergy = ApData.Energy.APenergyT / 3600 ;

	// cyclically trigger generation of Energy and DFT values on AP31x1
	if ( RBTrigDFT == TrigDFT )
	{
		TrigDFT ^= 1;
	}

	// Flat Stream Handling
	sFltRead.enable	 		= Flt_Enable;
	sFltRead.cfg		 	= fltMODE_FRAME;
	sFltRead.pBuf			= (UDINT)&TmpBuf[0];
	sFltRead.bufLen			= sizeof(TmpBuf);
	sFltRead.pRxBytes	 	= (UDINT)&FltMtuRd[0];
	sFltRead.rxBytesLen 	= sizeof(FltMtuRd);
	fltRead(&sFltRead);
	if (sFltRead.status == fltERR_FRAME_FINISHED)
	{
		if (sFltRead.validBytes - 1 == sizeof(X20AP31x1))
		{
			memcpy (&ApData, &TmpBuf[1], sizeof(X20AP31x1));
		}
	}

	sFltWrite.enable		= Flt_Enable;
	sFltWrite.cfg			= fltMODE_SYNCHRON + (1 << 4) + 2;
	sFltWrite.readSequ 		= sFltRead.readSequ;
	sFltWrite.pBuf			= (UDINT)&BlockNum;
	sFltWrite.bufLen	    = BlockAct;
	sFltWrite.pTxBytes		= (UDINT)&FltMtuWr[0];
	sFltWrite.txBytesLen	= sizeof(FltMtuWr);
	sFltWrite.pSequ	 		= (UDINT)&FltMtuRd[0];
	fltWrite(&sFltWrite);

} // end of  _CYCLIC
```

#### Test.var - Local variables
```iecst
(********************************************************************
 * COPYRIGHT -- Bernecker + Rainer
 ********************************************************************
 * Program: Test
 * File: Test.var
 * Author: wagnero
 * Created: May 11, 2011
 ********************************************************************
 * Local variables of program Test
 ********************************************************************)
VAR
	EnabEnergy : BOOL;
	FltMtuRd : ARRAY[0..30] OF USINT;
	FltMtuWr : ARRAY[0..30] OF USINT;
	RBTrigDFT : BOOL;
	TrigDFT : BOOL;
END_VAR
```

#### ApMap.h
```c
/* APMap.h - X20AP31x1 Data Mapping */
/*
------------------------------------------------------------------------------
 COPYRIGHT (C) BERNECKER + RAINER, AUSTRIA, A-5142 EGGELSBERG 120
------------------------------------------------------------------------------ */

/* == type definitions ====================================================	*/

typedef struct ADC_REG_STATUS	ADC_REG_STATUS;
struct ADC_REG_STATUS
{
	unsigned short 	SysStatus0;			// System Status 0
	unsigned short 	SysStatus1;			// System Status 1
	unsigned short 	EnStatus0;			// Metering Status 0
	unsigned short 	EnStatus1;			// Metering Status 1
};

typedef struct ADC_REG_RMS	ADC_REG_RMS;
struct ADC_REG_RMS
{
	unsigned short	IrmsN1;				// N Line Sampled current RMS
	unsigned short	UrmsA;				// phase A voltage RMS
	unsigned short	UrmsB;				// phase B voltage RMS
	unsigned short	UrmsC;				// phase C voltage RMS
	unsigned short	IrmsN0;				// N Line calculated current RMS
	unsigned short	IrmsA;				// phase A voltage RMS
	unsigned short	IrmsB;				// phase B voltage RMS
	unsigned short	IrmsC;				// phase C voltage RMS
};

typedef struct ADC_REG_THD_ANGLE	ADC_REG_THD_ANGLE;
struct ADC_REG_THD_ANGLE
{
//	THD+N, Frequency, Angle and Temperature Registers
	unsigned short	THDNUA;				// phase A voltage THD+N
	unsigned short	THDNUB;				// phase B voltage THD+N
	unsigned short	THDNUC;				// phase C voltage THD+N
	unsigned short	THDNIA;				// phase A current THD+N
	unsigned short	THDNIB;				// phase B current THD+N
	unsigned short	THDNIC;				// phase C current THD+N
	unsigned short	Freq;				// Frequency
	signed short	PAngleA;			// phase A mean phase angle
	signed short	PAngleB;			// phase B mean phase angle
	signed short	PAngleC;			// phase C mean phase angle
	signed short	Temp;				// Measured temperature
	signed short	UangleA;			// phase A voltage phase angle
	signed short	UangleB;			// phase B voltage phase angle
	signed short	UangleC;			// phase C voltage phase angle
};

typedef struct ADC_REG_POWER	ADC_REG_POWER;
struct ADC_REG_POWER
{
	unsigned short 	SVmeanTLSB;			// LSB of (Vector Sum) Total Apparent Power
	unsigned short 	SVmeanT;			// (Vector Sum) Total Apparent Power

// Power and Power Factor Register
	signed short	PmeanT;				// Total Active Power
	signed short	PmeanA;				// Phase A Active Power
	signed short	PmeanB;				// Phase B Active Power
	signed short	PmeanC;				// Phase C Active Power
	signed short	QmeanT;				// Total Reactive Power
	signed short	QmeanA;				// Phase A Reactive Power
	signed short	QmeanB;				// Phase B Reactive Power
	signed short	QmeanC;				// Phase C Reactive Power
	signed short	SAmeanT;			// (Arithmetic Sum) Total apparent power
	signed short	SmeanA;				// phase A apparent power
	signed short	SmeanB;				// phase B apparent power
	signed short	SmeanC;				// phase C apparent power
	signed short	PFmeanT;			// Total power factor
	signed short	PFmeanA;			// phase A power factor
	signed short	PFmeanB;			// phase B power factor
	signed short	PFmeanC;			// phase C power factor

// Fundamental/ Harmonic Power and Voltage/ Current RMS Registers
	signed short	PmeanTF;			// Total active fundamental power
	signed short	PmeanAF;			// phase A active fundamental power
	signed short	PmeanBF;			// phase B active fundamental power
	signed short	PmeanCF;			// phase C active fundamental power
	signed short	PmeanTH;			// Total active harmonic power
	signed short	PmeanAH;			// phase A active harmonic power
	signed short	PmeanBH;			// phase B active harmonic power
	signed short	PmeanCH;			// phase C active harmonic power
};

typedef struct ADC_REG_ENERGY	ADC_REG_ENERGY;
struct ADC_REG_ENERGY
{
	unsigned long 	APenergyT;			// Total Forward Active Energy
	unsigned long 	APenergyA;			// Phase A Forward Active Energy
	unsigned long 	APenergyB;			// Phase B Forward Active Energy
	unsigned long 	APenergyC;			// Phase C Forward Active Energy
	unsigned long 	ANenergyT;			// Total Reverse Active Energy
	unsigned long 	ANenergyA;			// Phase A Reverse Active Energy
	unsigned long 	ANenergyB;			// Phase B Reverse Active Energy
	unsigned long 	ANenergyC;			// Phase C Reverse Active Energy
	unsigned long 	RPenergyT;			// Total Forward Reactive Energy
	unsigned long 	RPenergyA;			// Phase A Forward Reactive Energy
	unsigned long 	RPenergyB;			// Phase B Forward Reactive Energy
	unsigned long 	RPenergyC;			// Phase C Forward Reactive Energy
	unsigned long 	RNenergyT;			// Total Reverse Reactive Energy
	unsigned long 	RNenergyA;			// Phase A Reverse Reactive Energy
	unsigned long 	RNenergyB;			// Phase B Reverse Reactive Energy
	unsigned long 	RNenergyC;			// Phase C Reverse Reactive Energy
	unsigned long 	SAenergyT;			// (Arithmetic Sum) Total Apparent Energy
	unsigned long 	SenergyA;		    // Phase A Apparent Energy
	unsigned long 	SenergyB;		   	// Phase B Apparent Energy
	unsigned long 	SenergyC;		    // Phase C Apparent Energy
	unsigned long 	SVenergyT;			// (Vector Sum) Total Apparent Energy

	// Fundamental / Harmonic Energy Register Register
	unsigned long 	APenergyTF;			// Total Forward Active Fundamental Energy
	unsigned long 	APenergyAF;			// Phase A Forward Active Fundamental Energy
	unsigned long 	APenergyBF;			// Phase B Forward Active Fundamental Energy
	unsigned long 	APenergyCF;			// Phase C Forward Active Fundamental Energy
	unsigned long 	ANenergyTF;			// Total Reverse Active Fundamental Energy
	unsigned long 	ANenergyAF;			// Phase A Reverse Active Fundamental Energy
	unsigned long 	ANenergyBF;			// Phase B Reverse Active Fundamental Energy
	unsigned long 	ANenergyCF;			// Phase C Reverse Active Fundamental Energy
	unsigned long 	APenergyTH;			// Total Forward Active Harmonic Energy
	unsigned long 	APenergyAH;			// Phase A Forward Active Harmonic Energy
	unsigned long 	APenergyBH;			// Phase B Forward Active Harmonic Energy
	unsigned long 	APenergyCH;			// Phase C Forward Active Harmonic Energy
	unsigned long 	ANenergyTH;			// Total Reverse Active Harmonic Energy
	unsigned long 	ANenergyAH;			// Phase A Reverse Active Harmonic Energy
	unsigned long 	ANenergyBH;			// Phase B Reverse Active Harmonic Energy
	unsigned long 	ANenergyCH;			// Phase C Reverse Active Harmonic Energy
	signed long		AEnergyT;			// Total Active Energy
	signed long 	REnergyT;			// Total Reactive Energy
};

typedef struct ADC_REG_DFT 	ADC_REG_DFT;
struct ADC_REG_DFT
{
	//	Arithmetic ratio, 2 bits integer and 14 bits fractional;	That is:	Harmonic Ratio (%) = Register Value / 163.84

	unsigned short	DftAI[32];		// phase A, Current, Harmonic Ratio for 2-th to 32-th order component and Total Harmonic Distortion	Ratio
	unsigned short	DftBI[32];		// phase B, Current, Harmonic Ratio for 2-th to 32-th order component and Total Harmonic Distortion	Ratio
	unsigned short	DftCI[32];		// phase C, Current, Harmonic Ratio for 2-th to 32-th order component and Total Harmonic Distortion	Ratio
	unsigned short	DftAV[32];		// phase A, Voltage, Harmonic Ratio for 2-th to 32-th order component and Total Harmonic Distortion	Ratio
	unsigned short	DftBV[32];		// phase B, Voltage, Harmonic Ratio for 2-th to 32-th order component and Total Harmonic Distortion	Ratio
	unsigned short	DftCV[32];		// phase C, Voltage, Harmonic Ratio for 2-th to 32-th order component and Total Harmonic Distortion	Ratio
	//	Format: Need special scaling/conversion.	The register value * 147.62 = full-scale input signal RMS.
	//	Current, Fundamental component value = Register Value * 209 * 65.535 / 8388608
	//	Voltage, Fundamental component value = Register Value * 209 * 655.35 / 8388608
	unsigned short	DftAI_Fund;
	unsigned short	DftAV_Fund;
	unsigned short	DftBI_Fund;
	unsigned short	DftBV_Fund;
	unsigned short	DftCI_Fund;
	unsigned short	DftCV_Fund;
};

typedef struct ADC_REG_CFGACT 	ADC_REG_CFGACT;
struct ADC_REG_CFGACT
{
	unsigned short  ChanControl;
	unsigned short  IDispTh;
	unsigned short  I_RatioA;
	unsigned short  I_RatioB;
	unsigned short  I_RatioC;
	unsigned short  I_RatioN;

	unsigned short  ZXConfig;
	unsigned short  SagTh;
	unsigned short  PhaseLoseTh;
	unsigned short  INWarnTh0;
	unsigned short  INWarnTh1;
	unsigned short  THDNUTh;
	unsigned short  THDNITh;
	unsigned short  MMode0;

	unsigned short 	PLconstL;
	unsigned short 	PLconstH;
};

typedef struct ENV_STATUS	ENV_STATUS;
struct ENV_STATUS
{
	unsigned long  ulUpTime;
	unsigned long  ulUpCnt;
	signed short   ssMinTemp;
	signed short   ssMaxTemp;
	unsigned long  ulRes[13];
};

typedef struct X20AP31x1	X20AP31x1;
struct X20AP31x1
{
	long					NetTimeReg;				// Time of Section copy to Buffer
	ADC_REG_STATUS			Status;  				// Status registers
	ADC_REG_RMS				Rms;	  			   	// RMS Registers
	ADC_REG_POWER			Power;				   	// Power Registers
	ADC_REG_THD_ANGLE		ThdAngle;			  	// THD + Angel Registers
	long				    NetTimeEnergy;			// Time of Section copy to Buffer
	ADC_REG_ENERGY			Energy;			      	// Energy Registers
	long				    NetTimeDft;			   	// Time of Section copy to Buffer
	ADC_REG_DFT				Dft;			       	// DFT Registers
	ADC_REG_CFGACT		    CfgAct;					// Config read back
	ENV_STATUS			    EnvReg;					// Read Back Environment Registers
};

#define ADC_BLK_ALL			    0
#define ADC_BLK_STATUS			1
#define ADC_BLK_RMS			    2
#define ADC_BLK_POWER		    3
#define ADC_BLK_THD_ANGLE		4
#define ADC_BLK_ENERGY			5
#define ADC_BLK_DFT			    6
#define ADC_BLK_CFGACT			7
#define ADC_BLK_ENVREG		    8
```

Listed in the project but not available here: Logical/Samples/GearAxis01/gearCyclic.st, Logical/Samples/GearAxis01/gear.typ
